TYPE ST_EL1809 :
STRUCT
	
	//Terminal 9
	bStartButton 										: BOOL;  // Term9_I.1 Start Button 
    bStopButton 										: BOOL;  // Term9_I.2 Stop Button 
    b24VPowerSupplyOK 									: BOOL;  // Term9_I.3 24V Power Supply OK 
    b24VPowerSupplyOKBck 								: BOOL;  // Term9_I.4 24V Power Supply OK Backup 
    b48VPowerSupplyOK 									: BOOL;  // Term9_I.5 48V Power Supply OK 
    bStageCollection_Home 								: BOOL;  // Term9_I.6 Stage Collection Home Position 
    bSampleRecovery_Vertical_Home 						: BOOL;  // Term9_I.7 Sample Recovery Vertical Home 
    bSampleRecovery_Horizontal_Home 					: BOOL;  // Term9_I.8 Sample Recovery Horizontal Home 
    bWasteOverflowSensor 								: BOOL;  // Term9_I.9 Waste Overflow Sensor 
    bUPSReady 											: BOOL;  // Term9_I.10 UPS Ready 
    bUPSReplaceBattery 									: BOOL;  // Term9_I.11 UPS Replace Battery 
    b48VPowerSupplyOKBck 								: BOOL;  // Term9_I.12 48V Us Power Supply OK 
    bCalibrationBoxPresent 								: BOOL;  // Term9_I.13 Calibration Box Present 
    bThroatJigPresent 									: BOOL;  // Term9_I.14 Throat Jig Present 

	//Terminal 30
	bAccessDoor4InterlockFdbk							: BOOL;  // Term30_I.1 Keyence Access Door Interlock Feedback
	bAccessDoor5InterlockFdbk							: BOOL;  // Term30_I.1 Keyence Access Door Interlock Feedback
	bAccessDoor6InterlockFdbk							: BOOL;  // Term30_I.1 Keyence Access Door Interlock Feedback

END_STRUCT
END_TYPE

(* stored: Version 1.1.0.1, ProductVersion 3.1.4024.15
   DUT ST_EL1809: Id {143ea90b-e3f2-482f-a224-3cd1f335b71e} *)
